FUNCTION_BLOCK FB_CoolingNetwork
VAR_INPUT
	//control struct for cn
	stCNControl : ST_CoolingNetworkControl;	
END_VAR
VAR_OUTPUT
	//temperatures in buffer storage
	fTemperatureBufferStorage : REAL;
END_VAR
VAR
	//systems
	BufferStorage : FB_BufferStorage;
	eChillerSystem : FB_eChillerSystem;
	HVFASystem : FB_HVFAStorageSystem;
	
	//internal variables
	fSetPoint_HVFASystem : REAL;
END_VAR

//buffer storage system
BufferStorage();
fTemperatureBufferStorage := BufferStorage.fMidTemperature;

//producer
eChillerSystem(bSetStatusOnAutomatic := stCNControl.bSetStatusOn_eChiller,
	bAlgorithmPermission := stCNControl.bAlgorithmPermission,
	fSetPointAutomatic := stCNControl.fTargetTemperature,
	fExternalTemperature := BufferStorage.fMidTemperature);
	
//external storages
//setpoint depends on loading mode -> storage must be cooler than setpoint temperature in network
IF stCNControl.bLoading_HVFASystem THEN
	fSetPoint_HVFASystem := stCNControl.fTargetTemperature-5;
ELSE
	fSetPoint_HVFASystem := stCNControl.fTargetTemperature;
END_IF
HVFASystem(bSetStatusOnAutomatic := stCNControl.bSetStatusOn_HVFASystem,
	bAlgorithmPermission := stCNControl.bAlgorithmPermission,
	fSetPointAutomatic := fSetpoint_HVFASystem,
	bLoadingAutomatic := stCNControl.bLoading_HVFASystem);

END_FUNCTION_BLOCK

(* stored: Version 1.1.0.1, ProductVersion 3.1.4024.10
   POU FB_CoolingNetwork: Id {3e3c7edc-aa3e-40d5-adb7-105c87a52325}, SpecialFunc None *)
